// TIA Portal V19 export
FUNCTION_BLOCK "TYPIC_C904_BF_VPI"   // FB42, FBD
TITLE = TYPIC_C904_BF_VPI: Vuilvloeistofpompinstallatie
{ S7_Optimized_Access := 'TRUE' }
AUTHOR : OCOTECH
FAMILY : Typical
NAME : C904.802
// Logisch Object Besturing: C904.802
// 
// Het doel van de BF VPI (vuilvloeistofpompinstallatie) is om de algemene sturing te voorzien van de vuilvloeistofpompinstallatie.
// 
// De algemene sturing omvat het weergeven van de algemene toestand en het aano en afschakelen van pompen in functie van het vloeistofpeil en het actieve regime.
// stored: MemoryReserve 10, SetENOAutomatically false
   VAR_INPUT
      CFG_TST_UTYD { ExternalAccessible := 'False'; ExternalVisible := 'False'; ExternalWritable := 'False'} : Time;   // Time-out standverandering pompinstallatie (transitiestatus onbereikt)
      CFG_TST_OK_TYD { ExternalAccessible := 'False'; ExternalVisible := 'False'; ExternalWritable := 'False'} : Time;   // Stabilisatietijd voor de toestand OK (bereikt)
      CFG_DEB_H { ExternalAccessible := 'False'; ExternalVisible := 'False'; ExternalWritable := 'False'} : Real;   // Grenswaarde minimaal debiet bij 1 aangeschakelde pomp
      CFG_ITYD_DEB { ExternalAccessible := 'False'; ExternalVisible := 'False'; ExternalWritable := 'False'} : Time;   // Tijdsvertraging voor alarm afvoer verstopt (pomp aangeschakeld en minimaal debiet niet bereikt)
      STU_CMD_AUT { ExternalAccessible := 'False'; ExternalVisible := 'False'; ExternalWritable := 'False'} : USInt;   // Groepscommando: schakel in automatisch
      STU_CMD_WRE { ExternalAccessible := 'False'; ExternalVisible := 'False'; ExternalWritable := 'False'} : USInt;   // Sturing regime
      STU_ALG_LCK_SIG { ExternalAccessible := 'False'; ExternalVisible := 'False'; ExternalWritable := 'False'} : USInt;   // Onderdruk alarmen
   END_VAR
   VAR_OUTPUT
      VAR_PWR { ExternalAccessible := 'False'; ExternalVisible := 'False'; ExternalWritable := 'False'} : Real;   // Som actuele vermogens van alle pompen
      STU_PMP1 { ExternalAccessible := 'False'; ExternalVisible := 'False'; ExternalWritable := 'False'} : USInt;   // Sturing pomp
      STU_PMP2 { ExternalAccessible := 'False'; ExternalVisible := 'False'; ExternalWritable := 'False'} : USInt;   // Sturing pomp
      STU_PMP3 { ExternalAccessible := 'False'; ExternalVisible := 'False'; ExternalWritable := 'False'} : USInt;   // Sturing pomp
      STU_IF_VPI { ExternalAccessible := 'False'; ExternalVisible := 'False'; ExternalWritable := 'False'} : USInt;   // Gewenst regime (naar interne sturing)
   END_VAR
   VAR_IN_OUT
      VAR_IF_VPI : "C904_VAR_IF_VPI_TYPIC";   // Struct met variabelen ontvangen van de interne sturing van de pompinstallatie
      VAR_PMP : Array[*] of "C904_VAR_PMP_TYPIC";   // Array met alle pompen, met alle variabelen van de pomp
      VAR_NIV : "C904_VAR_NIV_TYPIC";   // Struct met alle variabelen ontvangen van de subfunctie niveaumeting
      VAR_DEB : "C904_VAR_DEB_TYPIC";   // Struct met alle variabelen ontvangen van de subfunctie debietmeting
   END_VAR
   VAR
      BED : Struct   // Bedieningen
         ALG : Struct   // Gewenste stand
            X : "UDT_BED_ALG";
            KNOP { S7_SetPoint := 'True'} : Array[0..2] of "UDT_BED_KNOP";
         END_STRUCT;
      END_STRUCT;
      BED_ALG { ExternalWritable := 'False'} : "TYPIC_HF_BED_ALG_KNOP";   // Gewenste stand
      SIG { ExternalWritable := 'False'} : Struct   // Signaleringen
         AA01 : Bool;   // Gewenste stand niet bereikt (transitiestatus = niet bereikt)
         AA02 : Bool;   // Afvoer verstopt
         AB01 : Bool;   // Vuilvloeistofpompinstallatie niet beschikbaar
         AB02 : Bool;   // Vuilvloeistofpompinstallatie beperkt beschikbaar
      END_STRUCT;
      VAR { ExternalWritable := 'False'} : Struct   // Variabelen
         BSC : USInt;   // Geeft de beschikbaarheid aan van het deelsysteem
         TST_BWA : USInt;   // De status van de transitie van het deelsysteem
         BMO : USInt;   // Bedieningsmode
         WRE_BWA : USInt;   // Actueel regime
         CAPA : USInt;   // Beschikbare pompcapaciteit
         STS_NIV : USInt;   // Vloeistofniveau bepaald door de stand van de vlotters
         WRE_SWA { ExternalAccessible := 'False'; ExternalVisible := 'False'} : USInt;   // Gewenst regime
         REQ_AAN { ExternalAccessible := 'False'; ExternalVisible := 'False'} : USInt;   // Gewenst aantal aangeschakelde pompen
         CAPA_OK { ExternalAccessible := 'False'; ExternalVisible := 'False'} : USInt;   // Aantal beschikbare pompen
         STS_AAN { ExternalAccessible := 'False'; ExternalVisible := 'False'} : USInt;   // Actueel aantal aangeschakelde pompen
      END_STRUCT;
      HF_TST { ExternalAccessible := 'False'; ExternalVisible := 'False'; ExternalWritable := 'False'} : "TYPIC_HF_TST";   // Hulpfunctie transitiestatus
   END_VAR
   // // BED.ALG.KNOP[0] : Auto
   // // BED.ALG.KNOP[1] : Lozen
   // // BED.ALG.KNOP[2] : Uit
BEGIN

REGION Network 1: START
END_REGION

REGION Network 2: +++ Bedieningen +++
   // Vrijgave en verwerking van de bedieningen (centrale en lokale bediening). De bedienwaardes worden daarna in de verdere deelfunctionaliteiten gebruikt.
END_REGION

REGION Network 3: Knoppen BED_ALG(Gewenste stand)
   // Waardes en vrijge van de knoppen BED_ALG
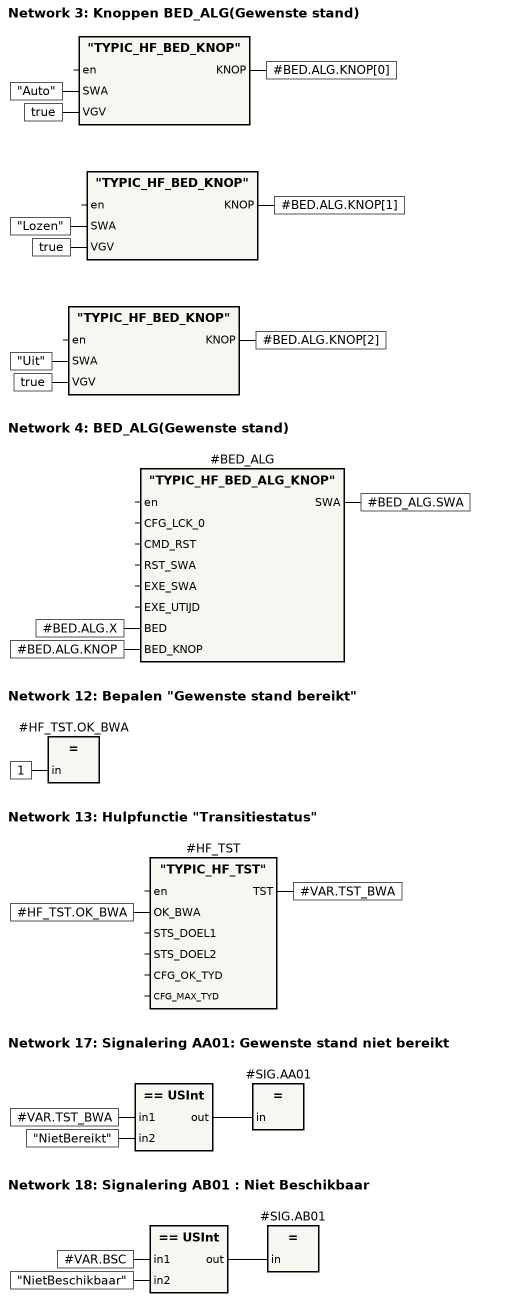
   "TYPIC_HF_BED_KNOP"(SWA := "Auto", VGV := true, KNOP => #BED.ALG.KNOP[0]);
   "TYPIC_HF_BED_KNOP"(SWA := "Lozen", VGV := true, KNOP => #BED.ALG.KNOP[1]);
   "TYPIC_HF_BED_KNOP"(SWA := "Uit", VGV := true, KNOP => #BED.ALG.KNOP[2]);
END_REGION

REGION Network 4: BED_ALG(Gewenste stand)
   // Verwerking BED_ALG
   #BED_ALG(BED := #BED.ALG.X, BED_KNOP := #BED.ALG.KNOP, SWA => #BED_ALG.SWA);   // "TYPIC_HF_BED_ALG_KNOP"
END_REGION

REGION Network 5: +++ Bepalen gewenst regime +++
   // Het gewenst regime (Lozen / Uit)
END_REGION

REGION Network 6: +++ Bepalen actueel regime en bedieningsmode +++
   // Bepalen bedieningsmode (Automatisch / Manueel / Hand) en daarna vastleggen van het actuele regime (Lozen / Uit).
END_REGION

REGION Network 7: +++ Berekeningen +++
   // Verscheidene berekeningen die nodig zijn voor de functionele werking of info voor weergave via de centrale en lokale bediening, zoals het aantal beschikbare pompen, het actueel aantal aangeschakelde pompen en de beschikbare pompcapaciteit.
END_REGION

REGION Network 8: +++ Bepalen vloeistofniveau +++
   // Het vloeistofniveau wordt bepaalt door, de status van de verschillende vlotters (ontvangen via de niveaumeting) en de vlotters droogloopbeveiliging van de pompen, om te zetten naar een status.
END_REGION

REGION Network 9: +++ Pompsturing bij regime “Uit” +++
   // Alle pompen behorende tot de schoonvloeistofinstallatie worden uitgeschakeld.
END_REGION

REGION Network 10: +++ Pompsturing bij regime “Lozen” +++
   // Pomp(en) aan- of uitschakelen op basis van de peilen LW en SW van de niveaumeting.
END_REGION

REGION Network 11: +++ Bepalen transitiestatus +++
   // Transitiestatus (bereikt / niet bereikt / in transitie) bepalen.
END_REGION

REGION Network 12: Bepalen "Gewenste stand bereikt"
   // Bepalen of de actuele stand in overeenstemming is met de gewenste stand
   #HF_TST.OK_BWA := 1;
END_REGION

REGION Network 13: Hulpfunctie "Transitiestatus"
   // De transitiestatus geeft de relatie tussen een gewenste stand (van een functionaliteit) en de actuele stand aan.
   #HF_TST(OK_BWA := #HF_TST.OK_BWA, TST => #VAR.TST_BWA);   // "TYPIC_HF_TST"
END_REGION

REGION Network 14: +++ Bepalen beschikbaarheidsstatus +++
   // Beschikbaarheidsstatus (beschikbaar / beperkt beschikbaar / niet beschikbaar) bepalen.
END_REGION

REGION Network 15 (SCL): Beschikbaarheidsstatus bepalen
   IF 
       //voorwaarden "Niet beschikbaar"
       TRUE
   THEN
       //Beschikbaarheidsstatus = Niet Beschikbaar
       #VAR.BSC:= "NietBeschikbaar";
   ELSIF
       //voorwaarden "Beperkt beschikbaar"
       TRUE
   THEN
       //Beschikbaarheidsstatus = Beperkt Beschikbaar
       #VAR.BSC:= "Beperkt";
   ELSE
       //Beschikbaarheidsstatus = Beschikbaar
       #VAR.BSC:= "Beschikbaar";
   END_IF;
END_REGION

REGION Network 16: +++ Signaleringen +++
   // Aanmaken signaleringen.
END_REGION

REGION Network 17: Signalering AA01: Gewenste stand niet bereikt
   #SIG.AA01 := #VAR.TST_BWA = "NietBereikt";
END_REGION

REGION Network 18: Signalering AB01 : Niet Beschikbaar
   #SIG.AB01 := #VAR.BSC = "NietBeschikbaar";
END_REGION

REGION Network 19: Signalering AB02 : Beperkt Beschikbaar
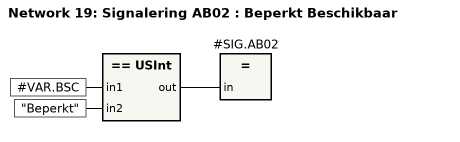
   #SIG.AB02 := #VAR.BSC = "Beperkt";
END_REGION

REGION Network 20: +++ Sturingen +++
   // Individuele commandos uitsturen naar iedere pomp om in- en uit te schakelen.
END_REGION

REGION Network 21: EINDE
   // Variabelen van intern scada rakvlak naar outputs copieren
END_REGION
END_FUNCTION_BLOCK
